FUNCTION F_PartIsClamped : BOOL
VAR_INPUT
	WX : sBogie;
END_VAR
VAR
END_VAR

IF (WX.A.bClamped AND WX.B.bClamped) OR NOT(WX.bEnabled) THEN
	F_PartIsClamped := 1;
	ELSE
		F_PartIsClamped := 0;
END_IF

END_FUNCTION

(* stored: Version 1.1.0.1, ProductVersion 3.1.4024.12
   POU F_PartIsClamped: Id {e822ac70-9b0f-43d9-a087-9cebb42b8f20}, SpecialFunc None *)
